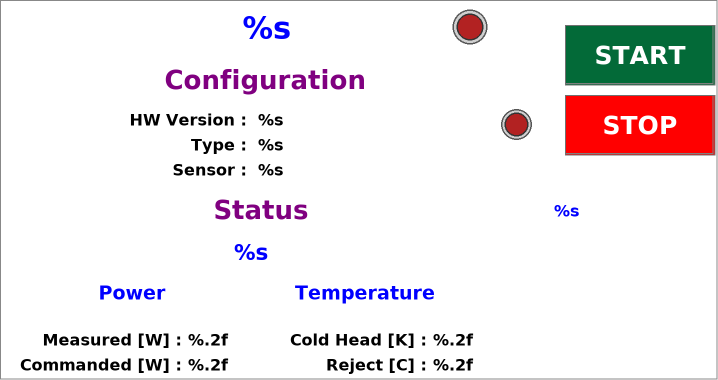
VISUALIZATION GUI_TEMPLATE_CRYOTELGT  // 718x380
VAR_IN_OUT
	m_Instance:	FB_CRYO_CRYOTELGT;
	m_bEnable:	BOOL;	// Flag to start/stop the cooler
END_VAR
    Rectangle (159,65 213x30), "Configuration"
    Rectangle (186,195 150x30), "Status"
    Rectangle (25,325 160x30), "Measured [W] :", tooltip "'P' command: Measured Power"
    Rectangle (185,325 70x30), "%.2f", text variable: m_Instance.stat.lrPowerMeasured
    Rectangle (152,10 230x36), "%s", text variable: m_Instance.in_sName
    Rectangle (255,155 110x30), "%s", text variable: m_Instance.stat.sSensor
    Rectangle (255,105 100x30), "%s", text variable: m_Instance.stat.sVersion
    Rectangle (255,130 100x30), "%s", text variable: m_Instance.stat.sMode
    Button (565,25 150x60), "START"
        OnMouseClick: execute { m_bEnable := TRUE; }
    Button (565,95 150x60), "STOP"
        OnMouseClick: execute { m_bEnable := FALSE; }
    Lamp1 (499,107 35x35), tooltip "If ON, there is a communication problem with the Cooler.", variable: m_Instance.bCommProblem, style: Lamp-Lamp1-Red
    Rectangle (36,235 431x35), "%s", tooltip "'COOLER' command: Cooler Control Mode: OFF or POWER", text variable: m_Instance.stat.sCtrlMode
    Rectangle (105,105 145x30), "HW Version :", tooltip "'VERSION' command: Current controller code version"
    Rectangle (105,130 145x30), "Type :", tooltip "'MODE' command: Cryocooler type, e.g. GT"
    Rectangle (105,155 145x30), "Sensor :", tooltip "'SENSOR' command: Configured temp. sensor type, e.g. 'PT-100'"
    Rectangle (57,278 150x30), "Power"
    Rectangle (290,278 150x30), "Temperature"
    Rectangle (25,350 160x30), "Commanded [W] :", tooltip "'PWOUT' command: Commanded power"
    Rectangle (185,350 70x30), "%.2f", text variable: m_Instance.stat.lrPowerCommanded
    Rectangle (285,325 145x30), "Cold Head [K] :", tooltip "'TC' command: Cold Head temperature"
    Rectangle (430,325 70x30), "%.2f", text variable: m_Instance.stat.lrTempColdHead
    Rectangle (285,350 145x30), "Reject [C] :", tooltip "'TEMP RJ' command: Reject Temperature"
    Rectangle (430,350 70x30), "%.2f", text variable: m_Instance.stat.lrTempReject
    Rectangle (416,196 302x30), "%s", tooltip "Cooler State", text variable: m_Instance.stat.sDevState
    Lamp1 (450,7 40x40), tooltip "If ON, Cooler is simulated.", variable: m_Instance.stat.bSimulation, invisible if: m_Instance.in_bSimulation = FALSE, style: Lamp-Lamp1-Red
END_VISUALIZATION

(* stored: Version 1.1.0.1, ProductVersion 3.1.4024.12
   Visu GUI_TEMPLATE_CRYOTELGT: Id {cb625138-2e21-43b0-b386-4895d985dd4e} *)
